FUNCTION GetSysTime : ULINT
VAR_INPUT
END_VAR
VAR
END_VAR

GetSysTime := Tc2_System.F_GetSystemTime() - 11644473600000000000;

END_FUNCTION

(* stored: Version 1.1.0.1
   POU GetSysTime: Id {9256dbe0-970c-46b2-beb0-50dc80b906e9}, SpecialFunc None *)
